Staubli VAL3: onStart.pgx

program onStart()
  local num i
  local bool bTest
begin
  // logMsg
  logMsg("[KERNEL] INTERFACE:PAGE Input Output")
  //
  sMode="OUT"
  sId=""
  nViewMode=0
  // refresh all
  call refreshStatic()
  call buildList(0)
  // record the old value....
  call use:selectNewField(nSelected,nIndex,nView)

end
